SUBAPPLICATION OneGeneratorOneConsumer_8_100x (* Subapplication Type *)
  (* Standard: 61499-2 *)
  (* Version 1.0, 2025-04-27, cochicde *)
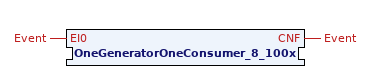
  EVENT_INPUT
    EI0;
  END_EVENT
  EVENT_OUTPUT
    CNF;
  END_EVENT
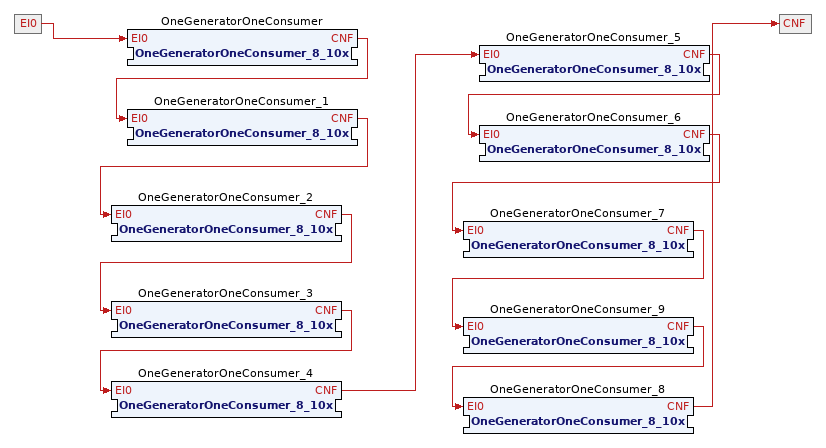
  SUBAPPS
    OneGeneratorOneConsumer : OneGeneratorOneConsumer_8_10x;
    OneGeneratorOneConsumer_1 : OneGeneratorOneConsumer_8_10x;
    OneGeneratorOneConsumer_2 : OneGeneratorOneConsumer_8_10x;
    OneGeneratorOneConsumer_3 : OneGeneratorOneConsumer_8_10x;
    OneGeneratorOneConsumer_4 : OneGeneratorOneConsumer_8_10x;
    OneGeneratorOneConsumer_5 : OneGeneratorOneConsumer_8_10x;
    OneGeneratorOneConsumer_6 : OneGeneratorOneConsumer_8_10x;
    OneGeneratorOneConsumer_7 : OneGeneratorOneConsumer_8_10x;
    OneGeneratorOneConsumer_8 : OneGeneratorOneConsumer_8_10x;
    OneGeneratorOneConsumer_9 : OneGeneratorOneConsumer_8_10x;
  END_SUBAPPS
  EVENT_CONNECTIONS
    OneGeneratorOneConsumer.CNF TO OneGeneratorOneConsumer_1.EI0;
    OneGeneratorOneConsumer_1.CNF TO OneGeneratorOneConsumer_2.EI0;
    OneGeneratorOneConsumer_2.CNF TO OneGeneratorOneConsumer_3.EI0;
    OneGeneratorOneConsumer_3.CNF TO OneGeneratorOneConsumer_4.EI0;
    OneGeneratorOneConsumer_6.CNF TO OneGeneratorOneConsumer_7.EI0;
    OneGeneratorOneConsumer_9.CNF TO OneGeneratorOneConsumer_8.EI0;
    OneGeneratorOneConsumer_5.CNF TO OneGeneratorOneConsumer_6.EI0;
    OneGeneratorOneConsumer_7.CNF TO OneGeneratorOneConsumer_9.EI0;
    OneGeneratorOneConsumer_4.CNF TO OneGeneratorOneConsumer_5.EI0;
    EI0 TO OneGeneratorOneConsumer.EI0;
    OneGeneratorOneConsumer_8.CNF TO CNF;
  END_CONNECTIONS
END_SUBAPPLICATION
